FUNCTION_BLOCK FB_PointManager EXTENDS FB_Utilities
VAR_INPUT
    {attribute 'OPC.UA.DA' := '1'}
    HMI_PM : stHMI_PM;
    pRobot : POINTER TO FB_1_ROB;
	MESSENGER: FB_Messenger;
	NameOfRobot : STRING := 'DUMMYROB';
END_VAR

VAR_OUTPUT
     nPointCount : UINT;
END_VAR

VAR
	editedPointPLC : stStoredPoint;	

    _sName         : STRING(80);
    _sDatabasePath : STRING(255);
    _bConfigured   : BOOL;

    // HMI command edges.
    _rNew       : R_TRIG;
    _rLoad      : R_TRIG;
    _rSave      : R_TRIG;
    _rDelete    : R_TRIG;
    _rTeach     : R_TRIG;
    _rSaveFile  : R_TRIG;
    _rLoadFile  : R_TRIG;
    _rMoveToEditedPoint : R_TRIG;
    _fMoveToEditedPoint : F_TRIG;

    _moveToEditedPointSettings : stCommand_Settings;
    _moveToEditedPointExecuteId : UINT;
    _moveToEditedPointPLC : stStoredPoint;

    // Editing identity. ID is kept privately so HMI writes can never change it.
    _nEditingId : DINT;
    _bEditingNew : BOOL;
    _nLastSelectedPointId : UDINT;
    _emptyPoint : stStoredPoint;

    // File state machines.
    _bReadFileActive  : BOOL;
    _bWriteFileActive : BOOL;
    _nLoadFileState : UINT;
    _nSaveFileState : UINT;
    _hLoadFile : UINT;
    _hSaveFile : UINT;

    _fileOpen  : FB_FileOpen;
    _fileRead  : FB_FileRead;
    _fileWrite : FB_FileWrite;
    _fileClose : FB_FileClose;

    // CSV is generated into/read from a byte buffer. This avoids STRING(255)
    // limitations for complete records/files.
    _csvWriter : FB_CSVMemBufferWriter;
    _csvReader : FB_CSVMemBufferReader;
    _fileBuffer : ARRAY[0..65535] OF BYTE;
    _nFileBufferSize : UDINT;
    _overflowByte : BYTE;

    // File data is validated here first and only committed to aPoints on success.
    _loadPoints : ARRAY[1..10] OF stStoredPoint;
    _nLoadPointCount : UINT;
	_Initialised: BOOL;
END_VAR



// HMI_PM is exposed as a two-way structure. Rebuild the fixed-size ComboBox
// source cyclically so stale client writes cannot restore duplicate zero IDs.
SyncPointList();

// Enforce immutable edit identity continuously, not only when SAVE is pressed.
IF (_nEditingId >= 1) AND (_nEditingId <= 10) THEN
    HMI_PM.editedPoint.id := _nEditingId;
END_IF



_rNew(CLK := HMI_PM.bCmdNew);
_rLoad(CLK := HMI_PM.bCmdLoad);
_rSave(CLK := HMI_PM.bCmdSave);
_rDelete(CLK := HMI_PM.bCmdDelete);
_rTeach(CLK := HMI_PM.bCmdTeach);
_rSaveFile(CLK := HMI_PM.bCmdSaveFile);
_rLoadFile(CLK := HMI_PM.bCmdLoadFile);
_rMoveToEditedPoint(CLK := HMI_PM.bMoveRobotToEditedPoint);
_fMoveToEditedPoint(CLK := HMI_PM.bMoveRobotToEditedPoint);

IF _fMoveToEditedPoint.Q THEN					//TODO
    IF (_moveToEditedPointExecuteId <> 0) AND (pRobot <> 0) THEN
		pRobot^.StopMotion();
    END_IF
    _moveToEditedPointExecuteId := 0;
END_IF

IF _rMoveToEditedPoint.Q THEN
    IF pRobot <> 0 THEN
        IF pRobot^.Operational
           AND (_nEditingId >= 1) AND (_nEditingId <= 10)
         AND ((HMI_PM.editedPoint.frame_id = eRefFrame.BRF)
             OR (HMI_PM.editedPoint.frame_id = eRefFrame.WRF)
             OR (HMI_PM.editedPoint.frame_id = eRefFrame.TRF)) THEN
//              OR (HMI_PM.editedPoint.frame_id = eRefFrame.CRF)) 

            _moveToEditedPointSettings.Name := HMI_PM.editedPoint.name;
            _moveToEditedPointSettings.Velocity := 50.0;
            _moveToEditedPointSettings.Acceleration := 500.0;
   
            _moveToEditedPointSettings.Target.frame_id := HMI_PM.editedPoint.frame_id;
            _moveToEditedPointPLC := PointFromHMI(Point := HMI_PM.editedPoint);
            _moveToEditedPointSettings.Target.pose.x := _moveToEditedPointPLC.x;
            _moveToEditedPointSettings.Target.pose.y := _moveToEditedPointPLC.y;
            _moveToEditedPointSettings.Target.pose.z := _moveToEditedPointPLC.z;
            _moveToEditedPointSettings.Target.pose.roll := _moveToEditedPointPLC.rx;
            _moveToEditedPointSettings.Target.pose.pitch := _moveToEditedPointPLC.ry;
            _moveToEditedPointSettings.Target.pose.yaw := _moveToEditedPointPLC.rz;

            _moveToEditedPointExecuteId := pRobot^.CommandHandler(
                Cmd := eCommands.MoveJ,
                Settings := _moveToEditedPointSettings
            );

            IF _moveToEditedPointExecuteId = 0 THEN
                HMI_PM.sLastOperation := 'Move to edited point was not accepted';
            ELSE
                HMI_PM.sLastOperation := 'Moving robot to edited point while button is held';
            END_IF
        ELSE
            _moveToEditedPointExecuteId := 0;
            HMI_PM.sLastOperation := 'Robot or edited point is not ready for motion';
        END_IF
    ELSE
        _moveToEditedPointExecuteId := 0;
        HMI_PM.sLastOperation := 'Robot or edited point is not ready for motion';
    END_IF
END_IF

// File operations own the manager until their asynchronous state machine finishes.
IF _bReadFileActive THEN
    LoadAllFromFile();
    RETURN;
END_IF

IF _bWriteFileActive THEN
    SaveAllToFile();
    RETURN;
END_IF

// Start file operations first so RAM data cannot be modified while a file is written/read.
IF _rLoadFile.Q THEN
    ;
    ;
    _bReadFileActive := TRUE;
    _nLoadFileState := 0;
    LoadAllFromFile();
    RETURN;
ELSIF _rSaveFile.Q THEN
    ;
    ;
    _bWriteFileActive := TRUE;
    _nSaveFileState := 0;
    SaveAllToFile();
    RETURN;
END_IF

// One RAM/edit operation per PLC cycle.
IF _rNew.Q THEN
    ;
    ;
    Create(sName := 'dummy', pose := HMI_PM.xCurrentTcp, frameId := eRefFrame.BRF);

ELSIF _rLoad.Q THEN
    ;
    ;
    IF (HMI_PM.nSelectedPointId >= 1) AND (HMI_PM.nSelectedPointId <= 10) THEN
        LoadById(nId := UDINT_TO_DINT(HMI_PM.nSelectedPointId));
    END_IF

ELSIF _rTeach.Q THEN
    ;
    ;
    Touchup(pose := HMI_PM.xCurrentTcp);

ELSIF _rSave.Q THEN
    ;
    ;
    Save();

ELSIF _rDelete.Q THEN
    ;
    ;
    IF (_nEditingId >= 1) AND (_nEditingId <= 10) THEN
        DeleteById(nId := _nEditingId);
    ELSIF (HMI_PM.nSelectedPointId >= 1) AND (HMI_PM.nSelectedPointId <= 10) THEN
        DeleteById(nId := UDINT_TO_DINT(HMI_PM.nSelectedPointId));
    ELSE
        ;
        MESSENGER.AddError(eMessageCategories.Undefined, CONCAT(NameOfRobot,' PM'), 'No point selected');
        
        
        HMI_PM.sLastOperation := 'No point selected';
    END_IF

ELSE
    // ComboBox SelectedId is the actual immutable point ID.
    // A changed selection loads the stored RAM value into both buffers.
    IF HMI_PM.nSelectedPointId <> _nLastSelectedPointId THEN
        _nLastSelectedPointId := HMI_PM.nSelectedPointId;

        IF (HMI_PM.nSelectedPointId >= 1) AND (HMI_PM.nSelectedPointId <= 10) THEN
            IF FindIndexById(nId := UDINT_TO_DINT(HMI_PM.nSelectedPointId)) <> 0 THEN
                ;
                ;
                LoadById(nId := UDINT_TO_DINT(HMI_PM.nSelectedPointId));
            END_IF
        END_IF
    END_IF
END_IF

METHOD PRIVATE AppendPointToSaveBuffer : BOOL
VAR_INPUT
    point : stStoredPoint;
END_VAR
AppendPointToSaveBuffer := FALSE;

IF NOT CsvPutField(sValue := DINT_TO_STRING(point.id), bFirst := FALSE, bEndRecord := FALSE) THEN RETURN; END_IF
IF NOT CsvPutField(sValue := point.name, bFirst := FALSE, bEndRecord := FALSE) THEN RETURN; END_IF
IF NOT CsvPutField(sValue := point.pose_kind, bFirst := FALSE, bEndRecord := FALSE) THEN RETURN; END_IF
IF NOT CsvPutField(sValue := DINT_TO_STRING(point.frame_id), bFirst := FALSE, bEndRecord := FALSE) THEN RETURN; END_IF
IF NOT CsvPutField(sValue := LREAL_TO_STRING(point.x), bFirst := FALSE, bEndRecord := FALSE) THEN RETURN; END_IF
IF NOT CsvPutField(sValue := LREAL_TO_STRING(point.y), bFirst := FALSE, bEndRecord := FALSE) THEN RETURN; END_IF
IF NOT CsvPutField(sValue := LREAL_TO_STRING(point.z), bFirst := FALSE, bEndRecord := FALSE) THEN RETURN; END_IF
IF NOT CsvPutField(sValue := LREAL_TO_STRING(point.rx), bFirst := FALSE, bEndRecord := FALSE) THEN RETURN; END_IF
IF NOT CsvPutField(sValue := LREAL_TO_STRING(point.ry), bFirst := FALSE, bEndRecord := FALSE) THEN RETURN; END_IF
IF NOT CsvPutField(sValue := LREAL_TO_STRING(point.rz), bFirst := FALSE, bEndRecord := FALSE) THEN RETURN; END_IF
IF NOT CsvPutField(sValue := 'mm_rad_v1', bFirst := FALSE, bEndRecord := TRUE) THEN RETURN; END_IF

AppendPointToSaveBuffer := TRUE;
END_METHOD

METHOD PRIVATE BuildSaveBuffer : BOOL
VAR
    i : UINT;
END_VAR
BuildSaveBuffer := FALSE;

// Tc2_Utilities CSV helper separator: force semicolon format.
DEFAULT_CSV_FIELD_SEP := 16#3B;

// Header. eEnumCmd_First resets/restarts the CSV memory writer.
IF NOT CsvPutField(sValue := 'id', bFirst := TRUE, bEndRecord := FALSE) THEN RETURN; END_IF
IF NOT CsvPutField(sValue := 'name', bFirst := FALSE, bEndRecord := FALSE) THEN RETURN; END_IF
IF NOT CsvPutField(sValue := 'pose_kind', bFirst := FALSE, bEndRecord := FALSE) THEN RETURN; END_IF
IF NOT CsvPutField(sValue := 'frame_id', bFirst := FALSE, bEndRecord := FALSE) THEN RETURN; END_IF
IF NOT CsvPutField(sValue := 'x', bFirst := FALSE, bEndRecord := FALSE) THEN RETURN; END_IF
IF NOT CsvPutField(sValue := 'y', bFirst := FALSE, bEndRecord := FALSE) THEN RETURN; END_IF
IF NOT CsvPutField(sValue := 'z', bFirst := FALSE, bEndRecord := FALSE) THEN RETURN; END_IF
IF NOT CsvPutField(sValue := 'rx', bFirst := FALSE, bEndRecord := FALSE) THEN RETURN; END_IF
IF NOT CsvPutField(sValue := 'ry', bFirst := FALSE, bEndRecord := FALSE) THEN RETURN; END_IF
IF NOT CsvPutField(sValue := 'rz', bFirst := FALSE, bEndRecord := FALSE) THEN RETURN; END_IF
IF NOT CsvPutField(sValue := 'unit_version', bFirst := FALSE, bEndRecord := TRUE) THEN RETURN; END_IF

FOR i := 1 TO nPointCount DO
    IF NOT AppendPointToSaveBuffer(point := HMI_PM.aPoints[i]) THEN
        RETURN;
    END_IF
END_FOR

_nFileBufferSize := _csvWriter.cbSize;
BuildSaveBuffer := TRUE;
END_METHOD

METHOD PRIVATE CheckName : BOOL
VAR_INPUT
    sInput    : STRING(80);
    nIgnoreId : DINT;
END_VAR
VAR
    i : UINT;
END_VAR
CheckName := FALSE;

IF sInput = '' THEN
    RETURN;
END_IF

IF NOT IsValidPointName(sValue := sInput) THEN
    RETURN;
END_IF

FOR i := 1 TO nPointCount DO
    IF (HMI_PM.aPoints[i].name = sInput)
       AND (HMI_PM.aPoints[i].id <> nIgnoreId) THEN
        RETURN;
    END_IF
END_FOR

CheckName := TRUE;
END_METHOD

METHOD PUBLIC Create : BOOL
VAR_INPUT
    sName   : STRING(80);
    pose    : ST_Pose;
    frameId : eRefFrame;
END_VAR
Create := PrepareNewPoint(
    sName := sName,
    pose := pose,
    frameId := frameId,
    sPoseKind := 'POSE_3D'
);
END_METHOD

METHOD PRIVATE CsvGetField : BOOL
VAR_INPUT
    bFirst : BOOL;
END_VAR
VAR_IN_OUT
    sValue     : STRING(255);
    bEndRecord : BOOL;
END_VAR
VAR
    sCsv : STRING(255);
END_VAR
CsvGetField := FALSE;
sValue := '';
bEndRecord := FALSE;

IF bFirst THEN
    _csvReader(
        eCmd := eEnumCmd_First,
        pBuffer := ADR(_fileBuffer),
        cbBuffer := _nFileBufferSize
    );
ELSE
    _csvReader(
        eCmd := eEnumCmd_Next,
        pBuffer := ADR(_fileBuffer),
        cbBuffer := _nFileBufferSize
    );
END_IF

IF NOT _csvReader.bOk THEN
    RETURN;
END_IF

sCsv := _csvReader.getValue;

// New files quote every field. Old unquoted files are accepted for migration.
IF (LEN(sCsv) >= 2) AND (LEFT(sCsv, 1) = '"') THEN
    sValue := CSVFIELD_TO_STRING(in := sCsv, bQM := TRUE);
ELSE
    sValue := CSVFIELD_TO_STRING(in := sCsv, bQM := FALSE);
END_IF

bEndRecord := _csvReader.bCRLF;
CsvGetField := TRUE;
END_METHOD

METHOD PRIVATE CsvPutField : BOOL
VAR_INPUT
    sValue     : STRING(255);
    bFirst     : BOOL;
    bEndRecord : BOOL;
END_VAR
VAR
    sCsv : STRING(255);
END_VAR
CsvPutField := FALSE;

// Point names reject CSV delimiters, so the writer can emit the documented plain format.
sCsv := STRING_TO_CSVFIELD(in := sValue, bQM := FALSE);

IF bFirst THEN
    _csvWriter(
        eCmd := eEnumCmd_First,
        putValue := sCsv,
        pValue := 0,
        cbValue := 0,
        bCRLF := bEndRecord,
        pBuffer := ADR(_fileBuffer),
        cbBuffer := SIZEOF(_fileBuffer)
    );
ELSE
    _csvWriter(
        eCmd := eEnumCmd_Next,
        putValue := sCsv,
        pValue := 0,
        cbValue := 0,
        bCRLF := bEndRecord,
        pBuffer := ADR(_fileBuffer),
        cbBuffer := SIZEOF(_fileBuffer)
    );
END_IF

CsvPutField := _csvWriter.bOk;
END_METHOD

METHOD PUBLIC DeleteById : BOOL
VAR_INPUT
    nId : DINT;
END_VAR
VAR
    nIndex      : UINT;
    nShiftIndex : UINT;
    nNextId     : DINT;
END_VAR
DeleteById := FALSE;

nIndex := FindIndexById(nId := nId);

IF nIndex = 0 THEN
    ;
    MESSENGER.AddError(eMessageCategories.Undefined, CONCAT(NameOfRobot,' PM'), 'Point ID not found');
    
    
    HMI_PM.sLastOperation := 'Point ID not found';
    RETURN;
END_IF

IF nIndex < nPointCount THEN
    FOR nShiftIndex := nIndex TO nPointCount - 1 DO
        HMI_PM.aPoints[nShiftIndex] := HMI_PM.aPoints[nShiftIndex + 1];
    END_FOR
END_IF

HMI_PM.aPoints[nPointCount] := _emptyPoint;
nPointCount := nPointCount - 1;

_nEditingId := 0;
_bEditingNew := FALSE;
HMI_PM.loadedPoint := _emptyPoint;
HMI_PM.editedPoint := _emptyPoint;



HMI_PM.nSelectedPointId := 0;
_nLastSelectedPointId := 0;
SyncPointList();

// Select and load the first remaining point, if any.
IF HMI_PM.nPointListCount > 0 THEN
    nNextId := UDINT_TO_DINT(HMI_PM.aPointList[1].id);
    LoadById(nId := nNextId);
END_IF

;
;


HMI_PM.sLastOperation := 'Deleted point from RAM array only';

DeleteById := TRUE;
END_METHOD

METHOD PRIVATE FindFreeId : DINT
VAR
    candidate : DINT;
    i         : UINT;
    bUsed     : BOOL;
END_VAR
FindFreeId := 0;

FOR candidate := 1 TO 10 DO
    bUsed := FALSE;

    FOR i := 1 TO nPointCount DO
        IF HMI_PM.aPoints[i].id = candidate THEN
            bUsed := TRUE;
            EXIT;
        END_IF
    END_FOR

    IF NOT bUsed THEN
        FindFreeId := candidate;
        RETURN;
    END_IF
END_FOR
END_METHOD

METHOD PRIVATE FindIndex : UINT
VAR_INPUT
    sName : STRING(80);
END_VAR
VAR
    i : UINT;
END_VAR
FindIndex := 0;

FOR i := 1 TO nPointCount DO
    IF HMI_PM.aPoints[i].name = sName THEN
        FindIndex := i;
        RETURN;
    END_IF
END_FOR
END_METHOD

METHOD PRIVATE FindIndexById : UINT
VAR_INPUT
    nId : DINT;
END_VAR
VAR
    i : UINT;
END_VAR
FindIndexById := 0;

IF (nId < 1) OR (nId > 10) THEN
    RETURN;
END_IF

FOR i := 1 TO nPointCount DO
    IF HMI_PM.aPoints[i].id = nId THEN
        FindIndexById := i;
        RETURN;
    END_IF
END_FOR
END_METHOD

METHOD PUBLIC Initialise : eResult
VAR_INPUT
    sName : STRING(80);
END_VAR
Initialise := NONE;

IF NOT IsValidDatabaseName(sValue := sName) THEN
    _bConfigured := FALSE;
    _sName := '';
    _sDatabasePath := '';
    ;
    MESSENGER.AddError(eMessageCategories.Undefined, CONCAT(NameOfRobot,' PM'), 'Invalid PointManager name for file path');
    
    
    HMI_PM.sLastOperation := 'Invalid PointManager name for file path';
    RETURN;
END_IF

_sName := sName;
_sDatabasePath := CONCAT('C:\Users\Public\Documents\', _sName);
_sDatabasePath := CONCAT(_sDatabasePath, '_saved_points.txt');
_bConfigured := TRUE;

;
;

HMI_PM.sLastOperation := 'Memory point store configured';

SyncPointList();
_Initialised:=TRUE;
Initialise := SUCCESS;
END_METHOD

METHOD PRIVATE IsValidDatabaseName : BOOL
VAR_INPUT
    sValue : STRING(80);
END_VAR
IsValidDatabaseName := FALSE;

IF (sValue = '') OR (sValue = '.') OR (sValue = '..') THEN
    RETURN;
END_IF

IF (FIND(sValue, '\') <> 0)
   OR (FIND(sValue, '/') <> 0)
   OR (FIND(sValue, ':') <> 0)
   OR (FIND(sValue, '*') <> 0)
   OR (FIND(sValue, '?') <> 0)
   OR (FIND(sValue, '"') <> 0)
   OR (FIND(sValue, '<') <> 0)
   OR (FIND(sValue, '>') <> 0)
   OR (FIND(sValue, '|') <> 0)
   OR (RIGHT(sValue, 1) = '.')
   OR (RIGHT(sValue, 1) = ' ') THEN
    RETURN;
END_IF

IsValidDatabaseName := TRUE;
END_METHOD

METHOD PRIVATE IsValidDintText : BOOL
VAR_INPUT
    sValue : STRING(255);
END_VAR
VAR
    i       : UINT;
    nLength : UINT;
    sChar   : STRING(1);
END_VAR
IsValidDintText := FALSE;
nLength := LEN(sValue);

IF nLength = 0 THEN
    RETURN;
END_IF

i := 1;
sChar := LEFT(sValue, 1);
IF (sChar = '+') OR (sChar = '-') THEN
    i := 2;
END_IF

IF i > nLength THEN
    RETURN;
END_IF

FOR i := i TO nLength DO
    sChar := MID(sValue, 1, i);
    IF (sChar < '0') OR (sChar > '9') THEN
        RETURN;
    END_IF
END_FOR

IsValidDintText := TRUE;
END_METHOD

METHOD PRIVATE IsValidLrealText : BOOL
VAR_INPUT
    sValue : STRING(255);
END_VAR
VAR
    i                    : UINT;
    nLength              : UINT;
    sChar                : STRING(1);
    bMantissaDigit       : BOOL;
    bDecimalPoint        : BOOL;
    bExponent            : BOOL;
    bExponentDigit       : BOOL;
    bExponentSignAllowed : BOOL;
END_VAR
IsValidLrealText := FALSE;
nLength := LEN(sValue);

IF nLength = 0 THEN
    RETURN;
END_IF

FOR i := 1 TO nLength DO
    sChar := MID(sValue, 1, i);

    IF (sChar >= '0') AND (sChar <= '9') THEN
        IF bExponent THEN
            bExponentDigit := TRUE;
            bExponentSignAllowed := FALSE;
        ELSE
            bMantissaDigit := TRUE;
        END_IF
    ELSIF (sChar = '+') OR (sChar = '-') THEN
        IF (i = 1) THEN
            // Leading sign is valid.
        ELSIF bExponentSignAllowed THEN
            bExponentSignAllowed := FALSE;
        ELSE
            RETURN;
        END_IF
    ELSIF sChar = '.' THEN
        IF bDecimalPoint OR bExponent THEN
            RETURN;
        END_IF
        bDecimalPoint := TRUE;
    ELSIF (sChar = 'E') OR (sChar = 'e') THEN
        IF bExponent OR NOT bMantissaDigit THEN
            RETURN;
        END_IF
        bExponent := TRUE;
        bExponentSignAllowed := TRUE;
    ELSE
        RETURN;
    END_IF
END_FOR

IsValidLrealText := bMantissaDigit AND (NOT bExponent OR bExponentDigit);
END_METHOD

METHOD PRIVATE IsValidPointName : BOOL
VAR_INPUT
        sValue : STRING(80);
END_VAR
IsValidPointName := (sValue <> '')
        AND (FIND(sValue, ';') = 0)
        AND (FIND(sValue, '"') = 0);
END_METHOD

METHOD PUBLIC Load : eResult
VAR_INPUT
    sName : STRING(80);
END_VAR
VAR
    nIndex : UINT;
END_VAR
Load := NONE;

nIndex := FindIndex(sName := sName);
IF nIndex = 0 THEN
    MESSENGER.AddError(eMessageCategories.Undefined, CONCAT(NameOfRobot,' PM'), 'Point name not found');
    
    
    HMI_PM.sLastOperation := 'Point name not found';
	Load := ERROR;
    RETURN;
END_IF

Load := LoadById(nId := HMI_PM.aPoints[nIndex].id);
END_METHOD

METHOD PUBLIC LoadAllFromFile : BOOL
VAR
    i : UINT;
    nFirstId : DINT;
END_VAR
LoadAllFromFile := FALSE;

CASE _nLoadFileState OF
    0:
        IF NOT _bConfigured THEN
            ;
            MESSENGER.AddError(eMessageCategories.Undefined, CONCAT(NameOfRobot,' PM'), 'PointManager name is not configured');
            
            
            HMI_PM.sLastOperation := 'PointManager name is not configured';
            _bReadFileActive := FALSE;
            RETURN;
        END_IF

        _nFileBufferSize := 0;
        _nLoadPointCount := 0;
        _fileOpen(bExecute := FALSE);
        _fileRead(bExecute := FALSE);
        _fileClose(bExecute := FALSE);
        _nLoadFileState := 10;
        RETURN;

    10:
        _fileOpen(
            sNetId := '',
            sPathName := _sDatabasePath,
            nMode := FOPEN_MODEREAD OR FOPEN_MODEBINARY,
            ePath := PATH_GENERIC,
            bExecute := TRUE,
            tTimeout := T#5S
        );

        IF _fileOpen.bBusy THEN RETURN; END_IF

        IF _fileOpen.bError THEN
            ;
            MESSENGER.AddError(eMessageCategories.Undefined, CONCAT(NameOfRobot,' PM'), 'File open for load failed');
            
            
            HMI_PM.sLastOperation := 'File open for load failed';
            _fileOpen(bExecute := FALSE);
            _nLoadFileState := 0;
            _bReadFileActive := FALSE;
            RETURN;
        END_IF

        _hLoadFile := _fileOpen.hFile;
        _fileOpen(bExecute := FALSE);
        _nLoadFileState := 20;
        RETURN;

    20:
        _fileRead(
            sNetId := '',
            hFile := _hLoadFile,
            pReadBuff := ADR(_fileBuffer),
            cbReadLen := SIZEOF(_fileBuffer),
            bExecute := TRUE,
            tTimeout := T#5S
        );

        IF _fileRead.bBusy THEN RETURN; END_IF

        IF _fileRead.bError THEN
            ;
            MESSENGER.AddError(eMessageCategories.Undefined, CONCAT(NameOfRobot,' PM'), 'File read failed');
            
            
            HMI_PM.sLastOperation := 'File read failed';
            _fileRead(bExecute := FALSE);
            _nLoadFileState := 30;
            RETURN;
        END_IF

        _nFileBufferSize := _fileRead.cbRead;
        _fileRead(bExecute := FALSE);

        // One extra byte read distinguishes an exactly-full buffer from an oversized file.
        _nLoadFileState := 25;
        RETURN;

    25:
        _fileRead(
            sNetId := '',
            hFile := _hLoadFile,
            pReadBuff := ADR(_overflowByte),
            cbReadLen := 1,
            bExecute := TRUE,
            tTimeout := T#5S
        );

        IF _fileRead.bBusy THEN RETURN; END_IF

        IF _fileRead.bError THEN
            ;
            MESSENGER.AddError(eMessageCategories.Undefined, CONCAT(NameOfRobot,' PM'), 'File size check failed');
            
            
            HMI_PM.sLastOperation := 'File size check failed';
        ELSIF _fileRead.cbRead > 0 THEN
            ;
            MESSENGER.AddError(eMessageCategories.Undefined, CONCAT(NameOfRobot,' PM'), 'Point file is larger than the PLC file buffer');
            
            
            HMI_PM.sLastOperation := 'Point file is larger than the PLC file buffer';
        END_IF

        _fileRead(bExecute := FALSE);
        _nLoadFileState := 30;
        RETURN;

    30:
        _fileClose(
            sNetId := '',
            hFile := _hLoadFile,
            bExecute := TRUE,
            tTimeout := T#5S
        );

        IF _fileClose.bBusy THEN RETURN; END_IF

        IF _fileClose.bError THEN
            ;
            MESSENGER.AddError(eMessageCategories.Undefined, CONCAT(NameOfRobot,' PM'), 'File close after load failed');
            
            
            HMI_PM.sLastOperation := 'File close after load failed';
        END_IF

        _fileClose(bExecute := FALSE);
        _hLoadFile := 0;


        _nLoadFileState := 40;
        RETURN;

    40:
        IF NOT ParseLoadBuffer() THEN
            _nLoadFileState := 0;
            _bReadFileActive := FALSE;
            RETURN;
        END_IF

        // Only now replace the live RAM array: the whole file has passed validation.
        FOR i := 1 TO 10 DO
            HMI_PM.aPoints[i] := _emptyPoint;
        END_FOR

        nPointCount := _nLoadPointCount;
        FOR i := 1 TO nPointCount DO
            HMI_PM.aPoints[i] := _loadPoints[i];
        END_FOR

        _nEditingId := 0;
        _bEditingNew := FALSE;
        HMI_PM.loadedPoint := _emptyPoint;
        HMI_PM.editedPoint := _emptyPoint;



        HMI_PM.nSelectedPointId := 0;
        _nLastSelectedPointId := 0;
        SyncPointList();

        IF HMI_PM.nPointListCount > 0 THEN
            nFirstId := UDINT_TO_DINT(HMI_PM.aPointList[1].id);
            LoadById(nId := nFirstId);
        END_IF

  
        HMI_PM.sLastOperation := 'Loaded and validated point file into RAM array';

        _nLoadFileState := 0;
        _bReadFileActive := FALSE;
        LoadAllFromFile := TRUE;
END_CASE
END_METHOD

METHOD PUBLIC LoadById : eResult
VAR_INPUT
    nId : DINT;
END_VAR
VAR
    nIndex : UINT;
END_VAR
LoadById := NONE;

nIndex := FindIndexById(nId := nId);

IF nIndex = 0 THEN
    MESSENGER.AddError(eMessageCategories.Undefined, CONCAT(NameOfRobot,' PM'), 'Point ID not found');
    HMI_PM.sLastOperation := 'Point ID not found';
	LoadById := ERROR;
    RETURN;
END_IF

// Stored RAM value is authoritative. Loading makes a fresh editable copy.
HMI_PM.loadedPoint := PointToHMI(Point := HMI_PM.aPoints[nIndex]);
HMI_PM.editedPoint := HMI_PM.loadedPoint;

_nEditingId := HMI_PM.loadedPoint.id;
_bEditingNew := FALSE;

// Protect ID even if HMI had previously written another value.
HMI_PM.editedPoint.id := _nEditingId;

HMI_PM.nSelectedPointId := DINT_TO_UDINT(_nEditingId);
_nLastSelectedPointId := HMI_PM.nSelectedPointId;


HMI_PM.sLastOperation := 'Loaded stored point into edit buffer';

LoadById := SUCCESS;
END_METHOD

PROPERTY LoadedPose : ST_Pose
GET
VAR
    Point : stStoredPoint;
END_VAR
Point := PointFromHMI(Point := HMI_PM.loadedPoint);
LoadedPose.x := Point.x;
LoadedPose.y := Point.y;
LoadedPose.z := Point.z;
LoadedPose.roll := Point.rx;
LoadedPose.pitch := Point.ry;
LoadedPose.yaw := Point.rz;
END_GET
END_PROPERTY

METHOD PRIVATE ParseLoadBuffer : BOOL
VAR
    sField     : STRING(255);
    bEnd       : BOOL;
    point      : stStoredPoint;
    nFrameId   : DINT;
    i          : UINT;
    j          : UINT;
    bLegacyUnits : BOOL;
END_VAR
ParseLoadBuffer := FALSE;
_nLoadPointCount := 0;

IF _nFileBufferSize = 0 THEN
    ;
    MESSENGER.AddError(eMessageCategories.Undefined, CONCAT(NameOfRobot,' PM'), 'Point file is empty');
    
    
    HMI_PM.sLastOperation := 'Point file is empty';
    RETURN;
END_IF

DEFAULT_CSV_FIELD_SEP := 16#3B;

// Header must exactly match the per-instance point database format.
IF NOT CsvGetField(bFirst := TRUE, sValue := sField, bEndRecord := bEnd) THEN
    SetFileParseError(); RETURN;
END_IF
IF (sField <> 'id') OR bEnd THEN SetFileParseError(); RETURN; END_IF

IF NOT CsvGetField(bFirst := FALSE, sValue := sField, bEndRecord := bEnd) THEN
    SetFileParseError(); RETURN;
END_IF
IF (sField <> 'name') OR bEnd THEN SetFileParseError(); RETURN; END_IF

IF NOT CsvGetField(bFirst := FALSE, sValue := sField, bEndRecord := bEnd) THEN
    SetFileParseError(); RETURN;
END_IF
IF (sField <> 'pose_kind') OR bEnd THEN SetFileParseError(); RETURN; END_IF

IF NOT CsvGetField(bFirst := FALSE, sValue := sField, bEndRecord := bEnd) THEN
    SetFileParseError(); RETURN;
END_IF
IF (sField <> 'frame_id') OR bEnd THEN SetFileParseError(); RETURN; END_IF

IF NOT CsvGetField(bFirst := FALSE, sValue := sField, bEndRecord := bEnd) THEN
    SetFileParseError(); RETURN;
END_IF
IF (sField <> 'x') OR bEnd THEN SetFileParseError(); RETURN; END_IF

IF NOT CsvGetField(bFirst := FALSE, sValue := sField, bEndRecord := bEnd) THEN
    SetFileParseError(); RETURN;
END_IF
IF (sField <> 'y') OR bEnd THEN SetFileParseError(); RETURN; END_IF

IF NOT CsvGetField(bFirst := FALSE, sValue := sField, bEndRecord := bEnd) THEN
    SetFileParseError(); RETURN;
END_IF
IF (sField <> 'z') OR bEnd THEN SetFileParseError(); RETURN; END_IF

IF NOT CsvGetField(bFirst := FALSE, sValue := sField, bEndRecord := bEnd) THEN
    SetFileParseError(); RETURN;
END_IF
IF (sField <> 'rx') OR bEnd THEN SetFileParseError(); RETURN; END_IF

IF NOT CsvGetField(bFirst := FALSE, sValue := sField, bEndRecord := bEnd) THEN
    SetFileParseError(); RETURN;
END_IF
IF (sField <> 'ry') OR bEnd THEN SetFileParseError(); RETURN; END_IF

IF NOT CsvGetField(bFirst := FALSE, sValue := sField, bEndRecord := bEnd) THEN
    SetFileParseError(); RETURN;
END_IF
IF sField <> 'rz' THEN SetFileParseError(); RETURN; END_IF

bLegacyUnits := bEnd;
IF NOT bLegacyUnits THEN
    IF NOT CsvGetField(bFirst := FALSE, sValue := sField, bEndRecord := bEnd) THEN
        SetFileParseError(); RETURN;
    END_IF
    IF (sField <> 'unit_version') OR NOT bEnd THEN SetFileParseError(); RETURN; END_IF
END_IF

WHILE TRUE DO
    point := _emptyPoint;

    // First field of next record. FALSE here after a complete CRLF-terminated record means EOF.
    IF NOT CsvGetField(bFirst := FALSE, sValue := sField, bEndRecord := bEnd) THEN
        EXIT;
    END_IF
    IF bEnd THEN SetFileParseError(); RETURN; END_IF
    IF NOT IsValidDintText(sValue := sField) OR (LEN(sField) > 2) THEN SetFileParseError(); RETURN; END_IF
    point.id := STRING_TO_DINT(sField);

    IF NOT CsvGetField(bFirst := FALSE, sValue := sField, bEndRecord := bEnd) THEN SetFileParseError(); RETURN; END_IF
    IF bEnd THEN SetFileParseError(); RETURN; END_IF
    IF NOT IsValidPointName(sValue := sField) THEN SetFileParseError(); RETURN; END_IF
    point.name := sField;

    IF NOT CsvGetField(bFirst := FALSE, sValue := sField, bEndRecord := bEnd) THEN SetFileParseError(); RETURN; END_IF
    IF bEnd THEN SetFileParseError(); RETURN; END_IF
    point.pose_kind := sField;

    IF NOT CsvGetField(bFirst := FALSE, sValue := sField, bEndRecord := bEnd) THEN SetFileParseError(); RETURN; END_IF
    IF bEnd THEN SetFileParseError(); RETURN; END_IF
    IF NOT IsValidDintText(sValue := sField) THEN SetFileParseError(); RETURN; END_IF
    nFrameId := STRING_TO_DINT(sField);
    CASE nFrameId OF
        0: point.frame_id := eRefFrame.BRF;
        1: point.frame_id := eRefFrame.WRF;
        2: point.frame_id := eRefFrame.TRF;
//         3: point.frame_id := eRefFrame.CRF;
        ELSE SetFileParseError(); RETURN;
    END_CASE

    IF NOT CsvGetField(bFirst := FALSE, sValue := sField, bEndRecord := bEnd) THEN SetFileParseError(); RETURN; END_IF
    IF bEnd THEN SetFileParseError(); RETURN; END_IF
    IF NOT IsValidLrealText(sValue := sField) THEN SetFileParseError(); RETURN; END_IF
    point.x := STRING_TO_LREAL(sField);

    IF NOT CsvGetField(bFirst := FALSE, sValue := sField, bEndRecord := bEnd) THEN SetFileParseError(); RETURN; END_IF
    IF bEnd THEN SetFileParseError(); RETURN; END_IF
    IF NOT IsValidLrealText(sValue := sField) THEN SetFileParseError(); RETURN; END_IF
    point.y := STRING_TO_LREAL(sField);

    IF NOT CsvGetField(bFirst := FALSE, sValue := sField, bEndRecord := bEnd) THEN SetFileParseError(); RETURN; END_IF
    IF bEnd THEN SetFileParseError(); RETURN; END_IF
    IF NOT IsValidLrealText(sValue := sField) THEN SetFileParseError(); RETURN; END_IF
    point.z := STRING_TO_LREAL(sField);

    IF NOT CsvGetField(bFirst := FALSE, sValue := sField, bEndRecord := bEnd) THEN SetFileParseError(); RETURN; END_IF
    IF bEnd THEN SetFileParseError(); RETURN; END_IF
    IF NOT IsValidLrealText(sValue := sField) THEN SetFileParseError(); RETURN; END_IF
    point.rx := STRING_TO_LREAL(sField);

    IF NOT CsvGetField(bFirst := FALSE, sValue := sField, bEndRecord := bEnd) THEN SetFileParseError(); RETURN; END_IF
    IF bEnd THEN SetFileParseError(); RETURN; END_IF
    IF NOT IsValidLrealText(sValue := sField) THEN SetFileParseError(); RETURN; END_IF
    point.ry := STRING_TO_LREAL(sField);

    IF NOT CsvGetField(bFirst := FALSE, sValue := sField, bEndRecord := bEnd) THEN SetFileParseError(); RETURN; END_IF
    IF NOT IsValidLrealText(sValue := sField) THEN SetFileParseError(); RETURN; END_IF
    point.rz := STRING_TO_LREAL(sField);

    IF bLegacyUnits THEN
        IF NOT bEnd THEN SetFileParseError(); RETURN; END_IF
        point.x := point.x * 1000.0;
        point.y := point.y * 1000.0;
        point.z := point.z * 1000.0;
    ELSE
        IF bEnd THEN SetFileParseError(); RETURN; END_IF
        IF NOT CsvGetField(bFirst := FALSE, sValue := sField, bEndRecord := bEnd) THEN SetFileParseError(); RETURN; END_IF
        IF (sField <> 'mm_rad_v1') OR NOT bEnd THEN SetFileParseError(); RETURN; END_IF
    END_IF

    IF (point.id < 1) OR (point.id > 10) THEN
        ;
        MESSENGER.AddError(eMessageCategories.Undefined, CONCAT(NameOfRobot,' PM'), 'File contains point ID outside 1..10');
        
        
        HMI_PM.sLastOperation := 'File contains point ID outside 1..10';
        RETURN;
    END_IF

    IF point.name = '' THEN
        ;
        MESSENGER.AddError(eMessageCategories.Undefined, CONCAT(NameOfRobot,' PM'), 'File contains an empty point name');
        
        
        HMI_PM.sLastOperation := 'File contains an empty point name';
        RETURN;
    END_IF

    IF (point.pose_kind <> 'POSE_2D') AND (point.pose_kind <> 'POSE_3D') THEN
        SetFileParseError();
        RETURN;
    END_IF

    // IDs are globally unique. Names are unique inside a robot prefix.
    FOR j := 1 TO _nLoadPointCount DO
        IF _loadPoints[j].id = point.id THEN
            ;
            MESSENGER.AddError(eMessageCategories.Undefined, CONCAT(NameOfRobot,' PM'), 'File contains duplicate point IDs');
            
            
            HMI_PM.sLastOperation := 'File contains duplicate point IDs';
            RETURN;
        END_IF

        IF _loadPoints[j].name = point.name THEN
            ;
            MESSENGER.AddError(eMessageCategories.Undefined, CONCAT(NameOfRobot,' PM'), 'File contains duplicate point names for one robot');
            
            
            HMI_PM.sLastOperation := 'File contains duplicate point names for one robot';
            RETURN;
        END_IF
    END_FOR

    IF _nLoadPointCount >= 10 THEN
        ;
        MESSENGER.AddError(eMessageCategories.Undefined, CONCAT(NameOfRobot,' PM'), 'File contains more than 10 points');
        
        
        HMI_PM.sLastOperation := 'File contains more than 10 points';
        RETURN;
    END_IF

    _nLoadPointCount := _nLoadPointCount + 1;
    _loadPoints[_nLoadPointCount] := point;
END_WHILE

ParseLoadBuffer := TRUE;
END_METHOD

METHOD PRIVATE PointFromHMI : stStoredPoint
VAR_INPUT
    Point : stStoredPoint;
END_VAR
PointFromHMI := Point;
PointFromHMI.x := ChangeRealFromHMIStandard(
    Value := Point.x, Category := eUnitCategory.Position);
PointFromHMI.y := ChangeRealFromHMIStandard(
    Value := Point.y, Category := eUnitCategory.Position);
PointFromHMI.z := ChangeRealFromHMIStandard(
    Value := Point.z, Category := eUnitCategory.Position);
PointFromHMI.rx := ChangeRealFromHMIStandard(
    Value := Point.rx, Category := eUnitCategory.Orientation);
PointFromHMI.ry := ChangeRealFromHMIStandard(
    Value := Point.ry, Category := eUnitCategory.Orientation);
PointFromHMI.rz := ChangeRealFromHMIStandard(
    Value := Point.rz, Category := eUnitCategory.Orientation);
END_METHOD

METHOD PRIVATE PointName : STRING(80)
VAR_INPUT
    sName : STRING(80);
    nId   : DINT;
END_VAR
IF sName <> '' THEN
    PointName := sName;
ELSE
    PointName := CONCAT('Point_', DINT_TO_STRING(nId));
END_IF
END_METHOD

METHOD PRIVATE PointToHMI : stStoredPoint
VAR_INPUT
    Point : stStoredPoint;
END_VAR
PointToHMI := Point;
PointToHMI.x := ChangeRealToHMIStandard(
    Value := Point.x, Category := eUnitCategory.Position);
PointToHMI.y := ChangeRealToHMIStandard(
    Value := Point.y, Category := eUnitCategory.Position);
PointToHMI.z := ChangeRealToHMIStandard(
    Value := Point.z, Category := eUnitCategory.Position);
PointToHMI.rx := ChangeRealToHMIStandard(
    Value := Point.rx, Category := eUnitCategory.Orientation);
PointToHMI.ry := ChangeRealToHMIStandard(
    Value := Point.ry, Category := eUnitCategory.Orientation);
PointToHMI.rz := ChangeRealToHMIStandard(
    Value := Point.rz, Category := eUnitCategory.Orientation);
END_METHOD

METHOD PRIVATE PrepareNewPoint : BOOL
VAR_INPUT
    sName     : STRING(80);
    pose      : ST_Pose;
    frameId   : eRefFrame;
    sPoseKind : STRING(16);
END_VAR
VAR
    nId : DINT;
END_VAR
PrepareNewPoint := FALSE;

IF nPointCount >= 10 THEN
    ;
    MESSENGER.AddError(eMessageCategories.Undefined, CONCAT(NameOfRobot,' PM'), 'Memory point store full');
    
    
    HMI_PM.sLastOperation := 'Memory point store full';
    RETURN;
END_IF

nId := FindFreeId();
IF nId = 0 THEN
    ;
    MESSENGER.AddError(eMessageCategories.Undefined, CONCAT(NameOfRobot,' PM'), 'No free point ID in range 1..10');
    
    
    HMI_PM.sLastOperation := 'No free point ID in range 1..10';
    RETURN;
END_IF

_nEditingId := nId;

_bEditingNew := TRUE;

// A new point is only an edit buffer until SAVE POINT is pressed.
HMI_PM.loadedPoint := _emptyPoint;
HMI_PM.editedPoint := _emptyPoint;

HMI_PM.editedPoint.id := _nEditingId;
HMI_PM.editedPoint.name := PointName(sName := sName, nId := _nEditingId);
HMI_PM.editedPoint.pose_kind := sPoseKind;
HMI_PM.editedPoint.frame_id := frameId;

HMI_PM.editedPoint.x := pose.x;
HMI_PM.editedPoint.y := pose.y;

IF sPoseKind = 'POSE_2D' THEN
    HMI_PM.editedPoint.z := 0;
    HMI_PM.editedPoint.rx := 0;
    HMI_PM.editedPoint.ry := 0;
    HMI_PM.editedPoint.rz := pose.yaw;
ELSE
    HMI_PM.editedPoint.z := pose.z;
    HMI_PM.editedPoint.rx := pose.roll;
    HMI_PM.editedPoint.ry := pose.pitch;
    HMI_PM.editedPoint.rz := pose.yaw;
END_IF

// Unsaved new point is not a stored selection yet.
// HMI_PM.nSelectedPointId := 0;
// _nLastSelectedPointId := 0;

MEMCPY(ADR(HMI_PM.aPoints[nId]),ADR(HMI_PM.editedPoint),SIZEOF(HMI_PM.editedPoint));
HMI_PM.editedPoint := PointToHMI(Point := HMI_PM.aPoints[nId]);


HMI_PM.nSelectedPointId := nId;
_nLastSelectedPointId := nId;
nPointCount := nPointCount +1;
HMI_PM.sLastOperation := 'New point ready for editing; press SAVE POINT to store it';

PrepareNewPoint := TRUE;
END_METHOD

METHOD PUBLIC Save : BOOL
Save := SaveEditedPoint();
END_METHOD

METHOD PUBLIC SaveAllToFile : BOOL
SaveAllToFile := FALSE;

CASE _nSaveFileState OF
    0:
        IF NOT _bConfigured THEN
            ;
            MESSENGER.AddError(eMessageCategories.Undefined, CONCAT(NameOfRobot,' PM'), 'PointManager name is not configured');
            
            
            HMI_PM.sLastOperation := 'PointManager name is not configured';
            _bWriteFileActive := FALSE;
            RETURN;
        END_IF

        IF NOT BuildSaveBuffer() THEN
            ;
            MESSENGER.AddError(eMessageCategories.Undefined, CONCAT(NameOfRobot,' PM'), 'Point file buffer overflow');
            
            
            HMI_PM.sLastOperation := 'Point file buffer overflow';
            _bWriteFileActive := FALSE;
            RETURN;
        END_IF

        _fileOpen(bExecute := FALSE);
        _fileWrite(bExecute := FALSE);
        _fileClose(bExecute := FALSE);
        _nSaveFileState := 10;
        RETURN;

    10:
        // FOPEN_MODEWRITE overwrites the existing file. No delete operation is used.
        _fileOpen(
            sNetId := '',
            sPathName := _sDatabasePath,
            nMode := FOPEN_MODEWRITE OR FOPEN_MODEBINARY,
            ePath := PATH_GENERIC,
            bExecute := TRUE,
            tTimeout := T#5S
        );

        IF _fileOpen.bBusy THEN RETURN; END_IF

        IF _fileOpen.bError THEN
            ;
            MESSENGER.AddError(eMessageCategories.Undefined, CONCAT(NameOfRobot,' PM'), 'File open for save failed');
            
            
            HMI_PM.sLastOperation := 'File open for save failed';
            _fileOpen(bExecute := FALSE);
            _nSaveFileState := 0;
            _bWriteFileActive := FALSE;
            RETURN;
        END_IF

        _hSaveFile := _fileOpen.hFile;
        _fileOpen(bExecute := FALSE);
        _nSaveFileState := 20;
        RETURN;

    20:
        _fileWrite(
            sNetId := '',
            hFile := _hSaveFile,
            pWriteBuff := ADR(_fileBuffer),
            cbWriteLen := _nFileBufferSize,
            bExecute := TRUE,
            tTimeout := T#5S
        );

        IF _fileWrite.bBusy THEN RETURN; END_IF

        IF _fileWrite.bError THEN
            ;
            MESSENGER.AddError(eMessageCategories.Undefined, CONCAT(NameOfRobot,' PM'), 'File write failed');
            
            
            HMI_PM.sLastOperation := 'File write failed';
        ELSIF _fileWrite.cbWrite <> _nFileBufferSize THEN
            ;
            MESSENGER.AddError(eMessageCategories.Undefined, CONCAT(NameOfRobot,' PM'), 'File write incomplete');
            
            
            HMI_PM.sLastOperation := 'File write incomplete';
        END_IF

        _fileWrite(bExecute := FALSE);
        _nSaveFileState := 30;
        RETURN;

    30:
        _fileClose(
            sNetId := '',
            hFile := _hSaveFile,
            bExecute := TRUE,
            tTimeout := T#5S
        );

        IF _fileClose.bBusy THEN RETURN; END_IF

        IF _fileClose.bError THEN
            ;
            MESSENGER.AddError(eMessageCategories.Undefined, CONCAT(NameOfRobot,' PM'), 'File close after save failed');
            
            
            HMI_PM.sLastOperation := 'File close after save failed';
        END_IF

        _fileClose(bExecute := FALSE);
        _hSaveFile := 0;
        _nSaveFileState := 0;
        _bWriteFileActive := FALSE;


        SaveAllToFile := TRUE;
        HMI_PM.sLastOperation := 'Overwrote point file with current RAM array';
END_CASE
END_METHOD

METHOD PUBLIC SaveEditedPoint : BOOL
VAR
    nIndex : UINT;
END_VAR
SaveEditedPoint := FALSE;

IF (_nEditingId < 1) OR (_nEditingId > 10) THEN
    ;
    MESSENGER.AddError(eMessageCategories.Undefined, CONCAT(NameOfRobot,' PM'), 'No valid edit point ID');
    
    
    HMI_PM.sLastOperation := 'No valid edit point ID';
    RETURN;
END_IF

IF NOT IsValidPointName(sValue := HMI_PM.editedPoint.name) THEN
    ;
    MESSENGER.AddError(eMessageCategories.Undefined, CONCAT(NameOfRobot,' PM'), 'Point name is empty or contains an invalid CSV character');
    
    
    HMI_PM.sLastOperation := 'Point name is empty or contains an invalid CSV character';
    RETURN;
END_IF

IF NOT CheckName(sInput := HMI_PM.editedPoint.name, nIgnoreId := _nEditingId) THEN
    ;
    MESSENGER.AddError(eMessageCategories.Undefined, CONCAT(NameOfRobot,' PM'), 'Point name already exists');
    
    
    HMI_PM.sLastOperation := 'Point name already exists';
    RETURN;
END_IF

// HMI is never authoritative for ID.
HMI_PM.editedPoint.id := _nEditingId;
editedPointPLC := PointFromHMI(Point := HMI_PM.editedPoint);
editedPointPLC.id := _nEditingId;

nIndex := FindIndexById(nId := _nEditingId);

IF nIndex = 0 THEN
    // New point: it only enters the RAM array here.
    IF NOT _bEditingNew THEN
        ;
        MESSENGER.AddError(eMessageCategories.Undefined, CONCAT(NameOfRobot,' PM'), 'Point ID is not present in RAM array');
        
        
        HMI_PM.sLastOperation := 'Point ID is not present in RAM array';
        RETURN;
    END_IF

    IF nPointCount >= 10 THEN
        ;
        MESSENGER.AddError(eMessageCategories.Undefined, CONCAT(NameOfRobot,' PM'), 'Memory point store full');
        
        
        HMI_PM.sLastOperation := 'Memory point store full';
        RETURN;
    END_IF

    nPointCount := nPointCount + 1;
    nIndex := nPointCount;

    // Metadata is created by the PLC, not by the HMI.
    HMI_PM.aPoints[nIndex].id := _nEditingId;
    HMI_PM.aPoints[nIndex].pose_kind := editedPointPLC.pose_kind;
    HMI_PM.aPoints[nIndex].frame_id := editedPointPLC.frame_id;
END_IF

// Existing point metadata and ID remain untouched.
// Only fields intended to be editable are committed.
HMI_PM.aPoints[nIndex].name := editedPointPLC.name;
HMI_PM.aPoints[nIndex].x := editedPointPLC.x;
HMI_PM.aPoints[nIndex].y := editedPointPLC.y;
HMI_PM.aPoints[nIndex].z := editedPointPLC.z;
HMI_PM.aPoints[nIndex].rx := editedPointPLC.rx;
HMI_PM.aPoints[nIndex].ry := editedPointPLC.ry;
HMI_PM.aPoints[nIndex].rz := editedPointPLC.rz;

// Reassert immutable identity after commit.
HMI_PM.aPoints[nIndex].id := _nEditingId;

// The newly stored RAM value becomes the read-only loaded version.
// Clear the edit buffer after SAVE POINT.
HMI_PM.loadedPoint := PointToHMI(Point := HMI_PM.aPoints[nIndex]);
HMI_PM.editedPoint := _emptyPoint;
_bEditingNew := FALSE;



HMI_PM.nSelectedPointId := DINT_TO_UDINT(_nEditingId);
_nLastSelectedPointId := HMI_PM.nSelectedPointId;
_nEditingId := 0;
SyncPointList();

;
;


HMI_PM.sLastOperation := 'Saved edited point to RAM array only';

SaveEditedPoint := TRUE;
END_METHOD

METHOD PRIVATE SetFileParseError
;
MESSENGER.AddError(eMessageCategories.Undefined, CONCAT(NameOfRobot,' PM'), 'Invalid or corrupt point file format');


HMI_PM.sLastOperation := 'Invalid or corrupt point file format';
END_METHOD

METHOD PRIVATE SyncPointList
VAR
    i              : UINT;
    nOutputIndex   : UINT;
    bSelectionSeen : BOOL;
    sText          : STRING(120);
END_VAR
HMI_PM.nPointListCount := 0;
bSelectionSeen := FALSE;

// ----------------------------------------------------------
// Initialize all ComboBox entries with unique placeholder IDs.
// This prevents duplicate id=0 errors in TcHmiCombobox.
// Placeholder IDs are 1001..1010.
// Real point IDs remain strictly 1..10.
// ----------------------------------------------------------
FOR i := 1 TO 10 DO
    HMI_PM.aPointList[i].id := 1000 + UINT_TO_UDINT(i);
    HMI_PM.aPointList[i].text := '';
    HMI_PM.aPointList[i].value := 0;
END_FOR


// ----------------------------------------------------------
// Fill active entries from this instance's stored point array.
// ----------------------------------------------------------
FOR i := 1 TO nPointCount DO
    HMI_PM.nPointListCount := HMI_PM.nPointListCount + 1;
    nOutputIndex := HMI_PM.nPointListCount;

    // Real point ID: always 1..10
    HMI_PM.aPointList[nOutputIndex].id :=
        DINT_TO_UDINT(HMI_PM.aPoints[i].id);

    HMI_PM.aPointList[nOutputIndex].value :=
        HMI_PM.aPoints[i].id;

        // Display text:
        // "ID 12 - PickPoint"
    sText := CONCAT(
        'ID ',
        DINT_TO_STRING(HMI_PM.aPoints[i].id)
    );

    sText := CONCAT(
        sText,
        ' - '
    );

    sText := CONCAT(
        sText,
        HMI_PM.aPoints[i].name
    );

    HMI_PM.aPointList[nOutputIndex].text := sText;


        // Check if current selection still exists.
    IF HMI_PM.nSelectedPointId =
        DINT_TO_UDINT(HMI_PM.aPoints[i].id)
    THEN
        bSelectionSeen := TRUE;
    END_IF
END_FOR


// ----------------------------------------------------------
// If the currently selected point no longer exists,
// select the first available point.
//
// 0 means "no selection" only.
// It is never a valid stored point ID.
// ----------------------------------------------------------
IF NOT bSelectionSeen THEN

    IF HMI_PM.nPointListCount > 0 THEN

        HMI_PM.nSelectedPointId :=
            HMI_PM.aPointList[1].id;

    ELSE

        HMI_PM.nSelectedPointId := 0;

    END_IF

END_IF
END_METHOD

METHOD PUBLIC Touchup : BOOL
VAR_INPUT
    pose : ST_Pose;
END_VAR
Touchup := FALSE;

IF (_nEditingId < 1) OR (_nEditingId > 10) THEN
    ;
    MESSENGER.AddError(eMessageCategories.Undefined, CONCAT(NameOfRobot,' PM'), 'No point loaded or prepared for editing');
    
    
    HMI_PM.sLastOperation := 'No point loaded or prepared for editing';
    RETURN;
END_IF

// ID is immutable. RETOUCH changes only the editable coordinates.
HMI_PM.editedPoint.id := _nEditingId;
HMI_PM.editedPoint.x := pose.x;
HMI_PM.editedPoint.y := pose.y;
HMI_PM.editedPoint.z := pose.z;
HMI_PM.editedPoint.rx := pose.roll;
HMI_PM.editedPoint.ry := pose.pitch;
HMI_PM.editedPoint.rz := pose.yaw;

HMI_PM.editedPoint := PointToHMI(Point := HMI_PM.editedPoint);

HMI_PM.sLastOperation := 'Current robot TCP copied to edited point only';

Touchup := TRUE;
END_METHOD

END_FUNCTION_BLOCK

(* stored: Version 1.1.0.1, ProductVersion 3.1.4026.18
   POU FB_PointManager: Id {9ded34ee-ef83-4142-8634-94e63622f962}, SpecialFunc None
   Method AppendPointToSaveBuffer: Id {02bde899-187e-49a8-8b98-6023034b73df}
   Method BuildSaveBuffer: Id {282801ee-e921-4c13-ac2e-f5915fe4b3c6}
   Method CheckName: Id {49a85f75-ccb9-4698-b4ad-70bfd4a1e615}
   Method Create: Id {2665e7b7-d388-4ca0-bb53-22244b7661b0}
   Method CsvGetField: Id {5e6f4a8b-cf59-4607-8e44-f9c41f24a2c4}
   Method CsvPutField: Id {c8f9b037-0b13-4e73-8ff6-6be8c41e92f1}
   Method DeleteById: Id {a41b206e-7a40-4611-9298-262c56c7c2f3}
   Method FindFreeId: Id {a382695d-4d70-4ad5-8f79-54f2e061e004}
   Method FindIndex: Id {b3052711-c116-4e8a-b375-f3f0fdea28de}
   Method FindIndexById: Id {c77c8bfa-3060-4d9d-8017-45f326721b38}
   Method Initialise: Id {09a6e83b-4d7f-41d5-944b-97ebdab99cae}
   Method IsValidDatabaseName: Id {b631ad6c-ae99-43ce-9480-cd5c79254916}
   Method IsValidDintText: Id {6cae7f0a-0988-4bd4-ae89-788a2cc15888}
   Method IsValidLrealText: Id {aa92088b-417c-4238-af93-e789fed2d3c1}
   Method IsValidPointName: Id {b0a74093-9fea-4747-b8b2-73a2068f3718}
   Method Load: Id {6d00c9c3-ae5f-47ac-82e1-a1471518898e}
   Method LoadAllFromFile: Id {4d27d444-7a0c-4a7c-a721-6aaa54255a19}
   Method LoadById: Id {434ff23f-8bbe-401c-84d5-3ced9c607a3b}
   Property LoadedPose: Id {ea20c9ff-92ea-4122-931a-45e49ef164f8}
   Get Get: Id {bf2f00be-2b86-46ea-90a3-3f38e1e8b036}
   Method ParseLoadBuffer: Id {02b12707-eafb-4400-96ec-be8eb15e5546}
   Method PointFromHMI: Id {9f000001-1111-2222-3333-000000000001}
   Method PointName: Id {ad3378e0-c724-4815-93f8-aff42bab454d}
   Method PointToHMI: Id {9f000001-1111-2222-3333-000000000002}
   Method PrepareNewPoint: Id {80738700-e5c4-418d-9db6-ba053e98625f}
   Method Save: Id {5ff36d6a-d948-4b70-adfa-e030735ba045}
   Method SaveAllToFile: Id {46482bb5-4a86-4095-81e3-f124bb50e79c}
   Method SaveEditedPoint: Id {77058650-029d-4f7d-b385-ecbe30b8cf36}
   Method SetFileParseError: Id {79872f9e-dca0-4435-99e7-fa1d894c9748}
   Method SyncPointList: Id {2e11b954-1e82-4a96-9fe4-24bc582a5e41}
   Method Touchup: Id {8f0ff160-e543-4f29-852c-514a30a0cc4a} *)
